PROGRAM AUTO
VAR
	//Stations
	Controller : RunUnitGeneric(argParent:= Controller, argSlotBase:= 0, argSlotLast:= 0);
	LifterCelluarA : ARRAY[1..3] OF RunLifterCelluar(argParent:= ADR(lifterCelluarA), 
									argSlotBase:= ADR(GVL.MATERIAL_SLOTS[1]), 
									argSlotLast:= ADR(GVL.MATERIAL_SLOTS[2]),
									argAxis:= ADR(GVL.axisControls[1]),
									argCylinder:=ADR(GVL.cylinderControls[1]),
									argHit:=ADR(GVL.commandBlocks[16]),
									argRelease:=ADR(GVL.commandBlocks[17]),
									argWorking:=ADR(GVL.commandBlocks[18]),		
									argObstacleSensor:= ADR(simuObstacleSensor),
									argReachSensor:= ADR(simuReachSensor));
	ConveyorMaster : RunUnitIndexerMasterCelluarA(argParent:= ADR(masterCelluarA), 
												argSlotBase:= ADR(GVL.MATERIAL_SLOTS[1]), 
												argSlotLast:= ADR(GVL.MATERIAL_SLOTS[2]),
												argAxis:=ADR(GVL.axisControls[2]),
												argUpstream:=ADR(masterProxy),		
												argCommandFast:=ADR(GVL.commandBlocks[32]),
												argCommandSlow:=ADR(GVL.commandBlocks[33]),
												argCommandTriggerRaise:=ADR(GVL.commandBlocks[40]),
												argCommandCheckRaise:=ADR(GVL.commandBlocks[41]));
	//
	nCounter : INT;
	bAllInitialized:BOOL;
	State : int;
END_VAR

IF NOT GVL.bObjectsInitialized THEN
	//all station initialize (build relationship) , machine spcific configuration
END_IF

CASE State OF
	0:
	bAllInitialized := TRUE;
	FOR nCounter:=1 TO 32 BY 1 DO
		IF gvl.stations[nCounter] <> 0 THEN
			gvl.stations[nCounter]^.Initialize();
		END_IF
		// if every station comes to 16#FF
		bAllInitialized := bAllInitialized AND (gvl.stations[nCounter]^.State = 16#FF);
	END_FOR
	1:
	//working
	FOR nCounter:=1 TO 32 BY 1 DO
		IF gvl.stations[nCounter] <> 0 THEN
			gvl.stations[nCounter]^();
		END_IF
		// if every station comes to 16#FF
		bAllInitialized := bAllInitialized AND (gvl.stations[nCounter]^.State = 16#FF);
	END_FOR
	//TODO , if initialize request raised , change to State-0
END_CASE

END_PROGRAM

(* stored: Version 1.1.0.1, ProductVersion 3.1.4022.10
   POU AUTO: Id {97a26fb9-68ff-461f-aa24-f8d33d7f3452}, SpecialFunc None *)
